TYPE ST_ENDURANCERUN_RECORD :
STRUCT
	id: DINT;
	dtTimeStamp: DT;
	sItem: STRING(255);
	diCycle: DINT;
	rWorkPressure: REAL;
	rLoadPressure: REAL;
	rPosition: REAL;
	rTemperature: REAL;
END_STRUCT
END_TYPE

(* stored: Version 1.1.0.1, ProductVersion 3.1.4024.12
   DUT ST_ENDURANCERUN_RECORD: Id {c5ae7290-156c-4cd6-855a-b6e867faac4f} *)
